// TIA Portal V20 export
VAR_GLOBAL   // PLC tag table "PROFIsafe Drives"
   BA010AZCRDR1_Status AT %I5100.0 : "safety.LDrvSafe_typeSinaTlg901Status";
   BA010AZCRDR1_Control AT %Q5100.0 : "safety.LDrvSafe_typeSinaTlg901Control";
   BA010AZCRDR2_Status AT %I5200.0 : "safety.LDrvSafe_typeSinaTlg901Status";
   BA010AZCRDR2_Control AT %Q5200.0 : "safety.LDrvSafe_typeSinaTlg901Control";
   BA010AZCRDR3_Status AT %I5300.0 : "safety.LDrvSafe_typeSinaTlg901Status";
   BA010AZCRDR3_Control AT %Q5300.0 : "safety.LDrvSafe_typeSinaTlg901Control";
   BA010AZCRDR4_Status AT %I5400.0 : "safety.LDrvSafe_typeSinaTlg901Status";
   BA010AZCRDR4_Control AT %Q5400.0 : "safety.LDrvSafe_typeSinaTlg901Control";
   BA010AZCRDR5_Status AT %I5500.0 : "safety.LDrvSafe_typeSinaTlg901Status";
   BA010AZCRDR5_Control AT %Q5500.0 : "safety.LDrvSafe_typeSinaTlg901Control";
   BA010AZCRDR6_Status AT %I5600.0 : "safety.LDrvSafe_typeSinaTlg901Status";
   BA010AZCRDR6_Control AT %Q5600.0 : "safety.LDrvSafe_typeSinaTlg901Control";
   BA010AZCRDR7_Status AT %I5700.0 : "safety.LDrvSafe_typeSinaTlg901Status";
   BA010AZCRDR7_Control AT %Q5700.0 : "safety.LDrvSafe_typeSinaTlg901Control";
   BA010AZCRDR8_Status AT %I5800.0 : "safety.LDrvSafe_typeSinaTlg901Status";
   BA010AZCRDR8_Control AT %Q5800.0 : "safety.LDrvSafe_typeSinaTlg901Control";
   BA010AZCRDR9_Status AT %I5900.0 : "safety.LDrvSafe_typeSinaTlg901Status";
   BA010AZCRDR9_Control AT %Q5900.0 : "safety.LDrvSafe_typeSinaTlg901Control";
   BA010AZCRDR10_Status AT %I6000.0 : "safety.LDrvSafe_typeSinaTlg901Status";
   BA010AZCRDR10_Control AT %Q6000.0 : "safety.LDrvSafe_typeSinaTlg901Control";
   BA010AZCRDR11_Status AT %I6100.0 : "safety.LDrvSafe_typeSinaTlg901Status";
   BA010AZCRDR11_Control AT %Q6100.0 : "safety.LDrvSafe_typeSinaTlg901Control";
   BA010AZCRDR12_Status AT %I6200.0 : "safety.LDrvSafe_typeSinaTlg901Status";
   BA010AZCRDR12_Control AT %Q6200.0 : "safety.LDrvSafe_typeSinaTlg901Control";
   BA010AZCRDR13_Status AT %I6300.0 : "safety.LDrvSafe_typeSinaTlg901Status";
   BA010AZCRDR13_Control AT %Q6300.0 : "safety.LDrvSafe_typeSinaTlg901Control";
   BA010AZCRDR14_Status AT %I6400.0 : "safety.LDrvSafe_typeSinaTlg901Status";
   BA010AZCRDR14_Control AT %Q6400.0 : "safety.LDrvSafe_typeSinaTlg901Control";
   BA010AZCRDR15_Status AT %I6500.0 : "safety.LDrvSafe_typeSinaTlg901Status";
   BA010AZCRDR15_Control AT %Q6500.0 : "safety.LDrvSafe_typeSinaTlg901Control";
   BA010AZCRDR16_Status AT %I9900.0 : "Safety.LDrvSafe_typeSinaGTlg30Status";
   BA010AZCRDR16_Control AT %Q9900.0 : "Safety.LDrvSafe_typeSinaGTlg30Control";
   BA010AZCRDR17_Status AT %I9918.0 : "Safety.LDrvSafe_typeSinaGTlg30Status";
   BA010AZCRDR17_Control AT %Q9918.0 : "Safety.LDrvSafe_typeSinaGTlg30Control";
   BA010AZCRDR18_Status AT %I9936.0 : "Safety.LDrvSafe_typeSinaGTlg30Status";
   BA010AZCRDR18_Control AT %Q9936.0 : "Safety.LDrvSafe_typeSinaGTlg30Control";
END_VAR
